% RSLogix 500 project project6.RSS, saved by version 8.30.00.16 %
PROJECT "UNTITLED"    % processor: Bul.1763 MicroLogix 1100 Series B %

PROGRAM FILES
  LAD 2 "MAIN"  13 rungs

DATA FILES
  O0 OUTPUT  4 elements
  I1 INPUT  6 elements
  S2 STATUS  66 elements
  B3 BINARY  2 elements
  T4 TIMER  4 elements
  C5 COUNTER  1 elements
  R6 CONTROL  1 elements
  N7 INTEGER  4 elements
  F8 FLOAT  1 elements

LADDER 2 "MAIN"
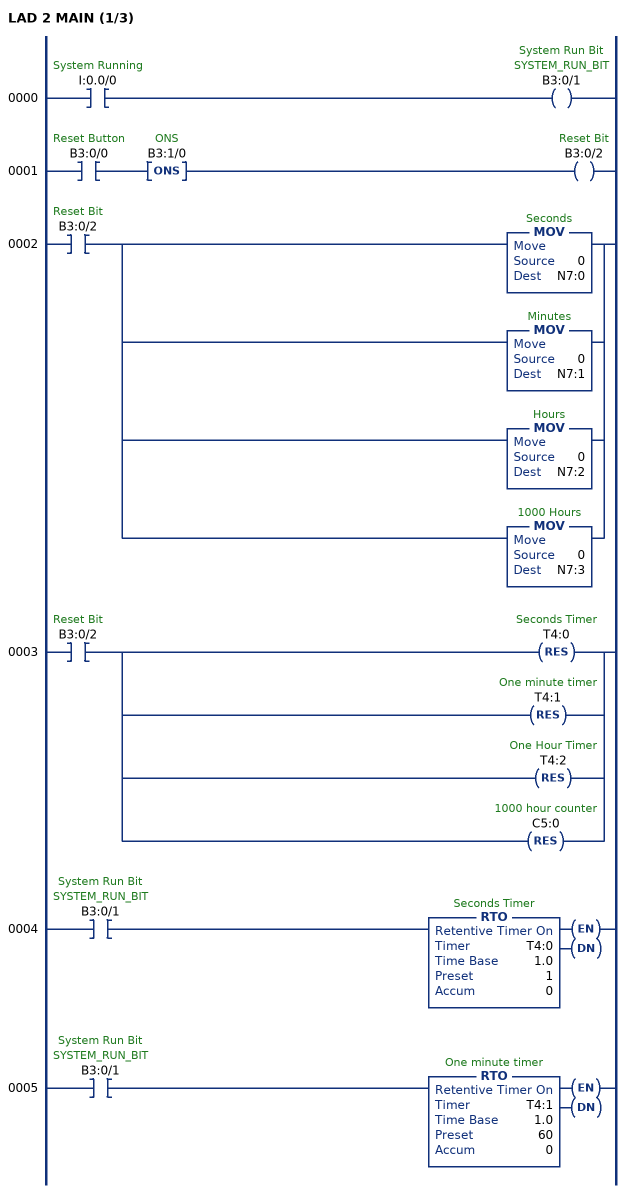
% Rung: 0 %
SOR XIC I:0.0/0 OTE B3:0/1 EOR
%   I:0.0/0  "System Running" %
%   B3:0/1  SYSTEM_RUN_BIT  "System Run Bit" %
% Rung: 1 %
SOR XIC B3:0/0 ONS B3:1/0 OTE B3:0/2 EOR
%   B3:0/0  "Reset Button" %
%   B3:1/0  "ONS" %
%   B3:0/2  "Reset Bit" %
% Rung: 2 %
SOR XIC B3:0/2 BST MOV 0 N7:0 NXB MOV 0 N7:1 NXB MOV 0 N7:2 NXB MOV 0 N7:3 BND EOR
%   B3:0/2  "Reset Bit" %
%   N7:0  "Seconds" %
%   N7:1  "Minutes" %
%   N7:2  "Hours" %
%   N7:3  "1000 Hours" %
% Rung: 3 %
SOR XIC B3:0/2 BST RES T4:0 NXB RES T4:1 NXB RES T4:2 NXB RES C5:0 BND EOR
%   B3:0/2  "Reset Bit" %
%   T4:0  "Seconds Timer" %
%   T4:1  "One minute timer" %
%   T4:2  "One Hour Timer" %
%   C5:0  "1000 hour counter" %
% Rung: 4 %
SOR XIC B3:0/1 RTO T4:0 1.0 1 0 EOR
%   B3:0/1  SYSTEM_RUN_BIT  "System Run Bit" %
%   T4:0  "Seconds Timer" %
% Rung: 5 %
SOR XIC B3:0/1 RTO T4:1 1.0 60 0 EOR
%   B3:0/1  SYSTEM_RUN_BIT  "System Run Bit" %
%   T4:1  "One minute timer" %

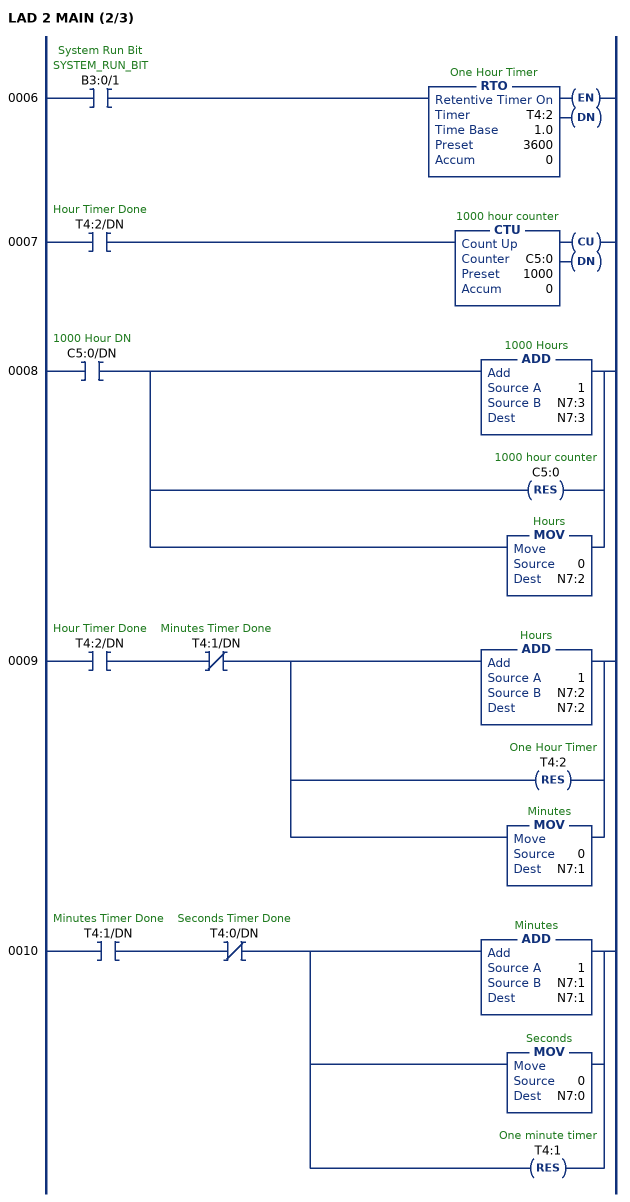
% Rung: 6 %
SOR XIC B3:0/1 RTO T4:2 1.0 3600 0 EOR
%   B3:0/1  SYSTEM_RUN_BIT  "System Run Bit" %
%   T4:2  "One Hour Timer" %
% Rung: 7 %
SOR XIC T4:2/DN CTU C5:0 1000 0 EOR
%   T4:2/DN  "Hour Timer Done" %
%   C5:0  "1000 hour counter" %
% Rung: 8 %
SOR XIC C5:0/DN BST ADD 1 N7:3 N7:3 NXB RES C5:0 NXB MOV 0 N7:2 BND EOR
%   C5:0/DN  "1000 Hour DN" %
%   N7:3  "1000 Hours" %
%   C5:0  "1000 hour counter" %
%   N7:2  "Hours" %
% Rung: 9 %
SOR XIC T4:2/DN XIO T4:1/DN BST ADD 1 N7:2 N7:2 NXB RES T4:2 NXB MOV 0 N7:1 BND EOR
%   T4:2/DN  "Hour Timer Done" %
%   T4:1/DN  "Minutes Timer Done" %
%   N7:2  "Hours" %
%   T4:2  "One Hour Timer" %
%   N7:1  "Minutes" %
% Rung: 10 %
SOR XIC T4:1/DN XIO T4:0/DN BST ADD 1 N7:1 N7:1 NXB MOV 0 N7:0 NXB RES T4:1 BND EOR
%   T4:1/DN  "Minutes Timer Done" %
%   T4:0/DN  "Seconds Timer Done" %
%   N7:1  "Minutes" %
%   N7:0  "Seconds" %
%   T4:1  "One minute timer" %

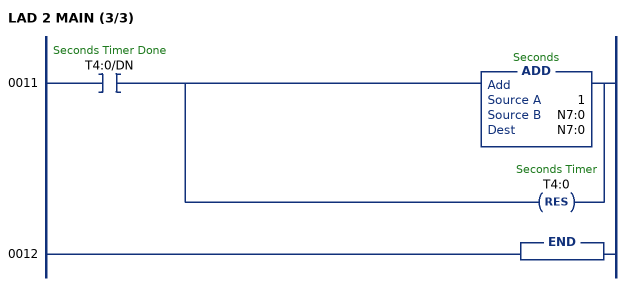
% Rung: 11 %
SOR XIC T4:0/DN BST ADD 1 N7:0 N7:0 NXB RES T4:0 BND EOR
%   T4:0/DN  "Seconds Timer Done" %
%   N7:0  "Seconds" %
%   T4:0  "Seconds Timer" %
% Rung: 12 %
SOR END EOR

OTHER DOCUMENTED ADDRESSES
  T4:3  "1000 hour timer"

DATA TABLE (non-zero values as saved)
DATA T4
% .PRE .ACC %
% T4:0 % 1 0
% T4:1 % 60 0
% T4:2 % 3600 0
DATA C5
% .PRE .ACC %
% C5:0 % 1000 0
